{attribute 'qualified_only'}
VAR_GLOBAL PERSISTENT
	parameter_Test:INT;
	parameter_Test_1:INT;
	parameter_Test_2:INT;
END_VAR

(* stored: Version 1.1.0.1, ProductVersion 3.1.4024.15
   GVL GVL_PERSISTENT: Id {db16c665-d563-455d-9463-d7926bcc8c88} *)
